{attribute 'GeneratedUsingTerminal: AMP8000-0030-0103-0103'}
{attribute addProperty BoxType "AMP8000-0030-0103-0103"}
{attribute addProperty Id "Safe_Logic_StateUSINT1Cycle_CounterUSINT1"}
{attribute addProperty CRC "331147839"}
{attribute addProperty Size "2"}
TYPE FSOE_13BCEA3F :
STRUCT
	{attribute addProperty Name "Safe_Logic_State"}
	Safe_Logic_State : USINT;
	{attribute addProperty Name "Cycle_Counter"}
	Cycle_Counter : USINT;
END_STRUCT
END_TYPE

(* stored: Version 1.2.0.0, ProductVersion 3.1.4024.9
   DUT FSOE_13BCEA3F: Id {9b5232ec-fe2e-426a-98f7-2a448a0a653b} *)
